% RSLogix 500 project PROJECT5.RSS, saved by version 8.30.00.16 %
PROJECT "PROJECT5"    % processor: Bul.1763 MicroLogix 1100 Series B %

PROGRAM FILES
  LAD 2 "MAIN"  3 rungs

DATA FILES
  O0 OUTPUT  5 elements
  I1 INPUT  7 elements
  S2 STATUS  66 elements
  B3 BINARY  1 elements
  T4 TIMER  1 elements
  C5 COUNTER  1 elements
  R6 CONTROL  1 elements
  N7 INTEGER  1 elements
  F8 FLOAT  1 elements

LADDER 2 "MAIN"
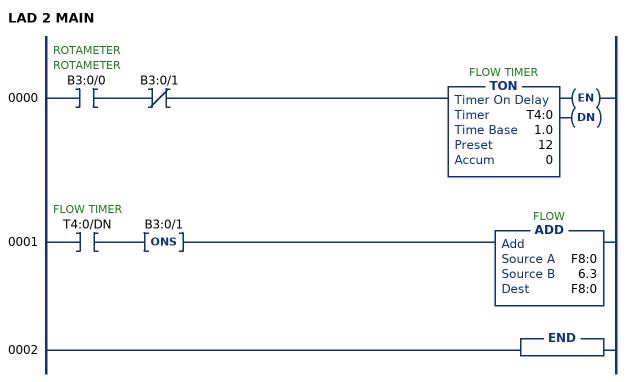
% Rung: 0 %
SOR XIC B3:0/0 XIO B3:0/1 TON T4:0 1.0 12 0 EOR
%   B3:0/0  ROTAMETER  "ROTAMETER" %
%   T4:0  "FLOW TIMER" %
% Rung: 1 %
SOR XIC T4:0/DN ONS B3:0/1 ADD F8:0 6.3 F8:0 EOR
%   T4:0  "FLOW TIMER" %
%   F8:0  "FLOW" %
% Rung: 2 %
SOR END EOR

DATA TABLE (non-zero values as saved)
DATA T4
% .PRE .ACC %
% T4:0 % 12 0
